Omron CX-Programmer project NewProject (CX-Programmer 9.75)

# PLC Project2: CP1L M

## Global symbols (name address type ; comment)
0.00 BOOL  ; PB_Start
0.01 BOOL  ; PB_Stop
100.00 BOOL  ; Lamp 1
100.01 BOOL  ; Lamp 2
200.00 BOOL  ; IR 1

## Program NewProgram1 (cyclic task 0)

### Section Section1

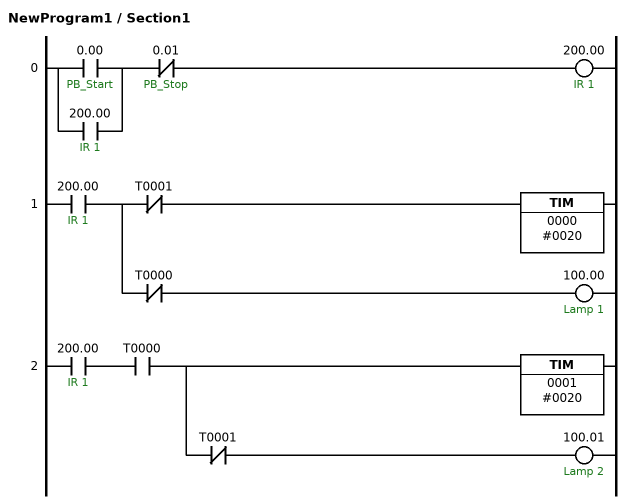
; rung 0
LD 0.00  ; PB_Start
OR 200.00  ; IR 1
ANDNOT 0.01  ; PB_Stop
OUT 200.00  ; IR 1
; rung 1
LD 200.00  ; IR 1
OUT TR0
ANDNOT T0001
TIM 0000 #0020
LD TR0
ANDNOT T0000
OUT 100.00  ; Lamp 1
; rung 2
LD 200.00  ; IR 1
AND T0000
TIM 0001 #0020
ANDNOT T0001
OUT 100.01  ; Lamp 2

### Section END
; rung 0
END(001)